(* Logix 5000 project; controller Hose_HP_Test_Rig_V1 vendor 1 type 14 code 149 rev 32.11; software revision 32.00; part 10 of 10 *)
(* tags used below, declared in another part *)
   INDV_LTEST_ON_STN4 : BOOL;
   ONS104 : BOOL;
   ONS4 : BOOL;
   TEST_INIT_DEL_STN4 : TIMER;
   AUTO_DOOR_OPEN_SEQ_STN4 : DINT;
   AUTO_TEST_ON_STN4 : BOOL;
   BOTTOM_CLAMP_SEQ_STN4 : DINT;
   BOTTOM_DECLAMP_SEQ_STN4 : DINT;
   CLR_ONS_STN4 : BOOL;
   CONS_CALB_ON_STN4 : BOOL;
   CONS_STS_STN1 : DINT;
   CONS_STS_STN2 : DINT;
   CONS_STS_STN3 : DINT;
   CONS_STS_STN4 : DINT;
   CONS_TEST_ON : BOOL;
   CYCLE_TIME_ACT_STN4 : REAL;
   DUMMIT : BOOL;
   FAIL_COUNT_RETEST : DINT;
   FAIL_COUNT_RETEST_STN2 : DINT;
   FAULTED_STN1 : BOOL;
   FAULTED_STN2 : BOOL;
   FAULTED_STN3 : BOOL;
   FAULTED_STN4 : BOOL;
   FP_ACCESS_OK : ALIAS FOR Local:2:I.Data.24;
   HP_SENSOR_SEL : BOOL;
   HP_STS_STN1 : DINT;
   HP_STS_STN2 : DINT;
   HP_STS_STN3 : DINT;
   HP_STS_STN4 : DINT;
   HP_TEST_ON : BOOL;
   INDV_CTEST_ON_STN4 : BOOL;
   INIT_STN4 : BOOL;
   MAIN_MENU : BOOL;
   MAIN_MENU_OFF : TIMER;
   OTHER_SENSOR_SEL : BOOL;
   PASS_COUNT_RETEST : DINT;
   PASS_COUNT_RETEST_STN2 : DINT;
   PASSED_STN4 : BOOL;
   PASSWORD_SET : DINT;
   RETEST : BOOL;
   RETEST_FAIL_COUNT : DINT;
   RETEST_ON_PROHIBIT : BOOL;
   RETEST_PASS_COUNT : DINT;
   RETEST_SET_COUNT : DINT;
   SCR_STS : DINT[6];
   SENS_CAL_SEL_BOTTOM_CLAMP : BOOL;
   SENS_CAL_SEL_MASTER : BOOL;
   SENS_CAL_SEL_STAMP : BOOL;
   SENS_CAL_SEL_TOP_CLAMP : BOOL;
   SENS_CALB_SEL_STN1 : BOOL;
   SENS_CALB_SEL_STN2 : BOOL;
   SENS_CALB_SEL_STN3 : BOOL;
   SENS_CALB_SEL_STN4 : BOOL;
   SEQ_NO_STN4 : DINT;
   STN1_TEST_STS : DINT;
   STN2_TEST_STS : DINT;
   STN3_TEST_STS : DINT;
   STN4_TEST_STS : DINT;
   STS : DINT;
   STS_OP_STN4 : DINT;
   TEST_ON_STN4 : BOOL;
   TOP_CLAMP_SEQ_STN4 : DINT;
   TS_STS_STN4 : DINT;
   USER_CHG : TIMER;
   VIEW_PARAM : BOOL;
   VIEW_PARAM_OFF : TIMER;
   WHICH_USER : INT;
(* MainProgram, continued *)

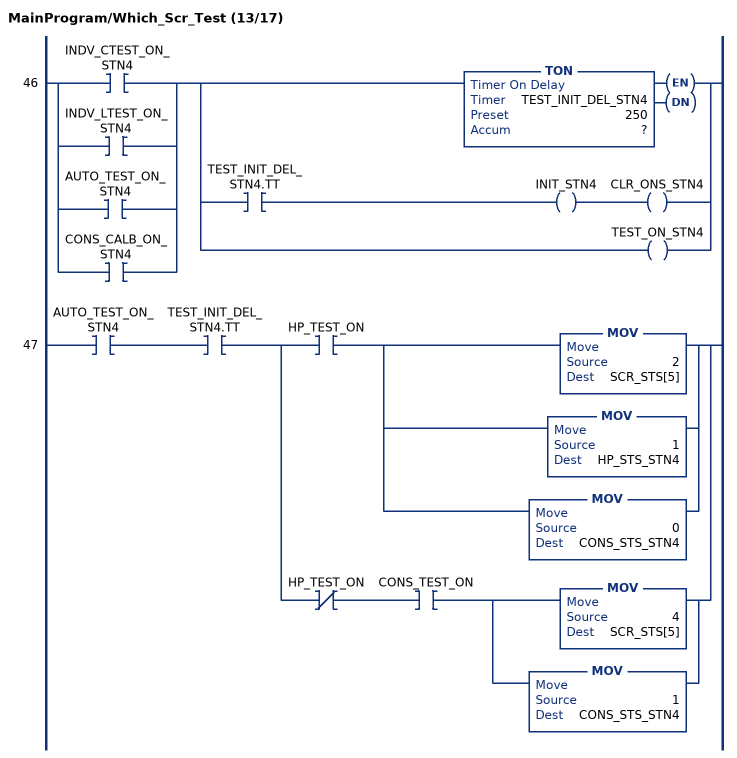
   [picture p174: MainProgram/Which_Scr_Test rungs 46-47]
   46: [XIC(INDV_CTEST_ON_STN4) ,XIC(INDV_LTEST_ON_STN4) ,XIC(AUTO_TEST_ON_STN4) ,XIC(CONS_CALB_ON_STN4) ][TON(TEST_INIT_DEL_STN4,?,?) ,XIC(TEST_INIT_DEL_STN4.TT) OTE(INIT_STN4) OTE(CLR_ONS_STN4) ,OTE(TEST_ON_STN4) ];
   47: XIC(AUTO_TEST_ON_STN4)XIC(TEST_INIT_DEL_STN4.TT)[XIC(HP_TEST_ON) [MOV(2,SCR_STS[5]) ,MOV(1,HP_STS_STN4) ,MOV(0,CONS_STS_STN4) ] ,XIO(HP_TEST_ON) XIC(CONS_TEST_ON) [MOV(4,SCR_STS[5]) ,MOV(1,CONS_STS_STN4) ] ];
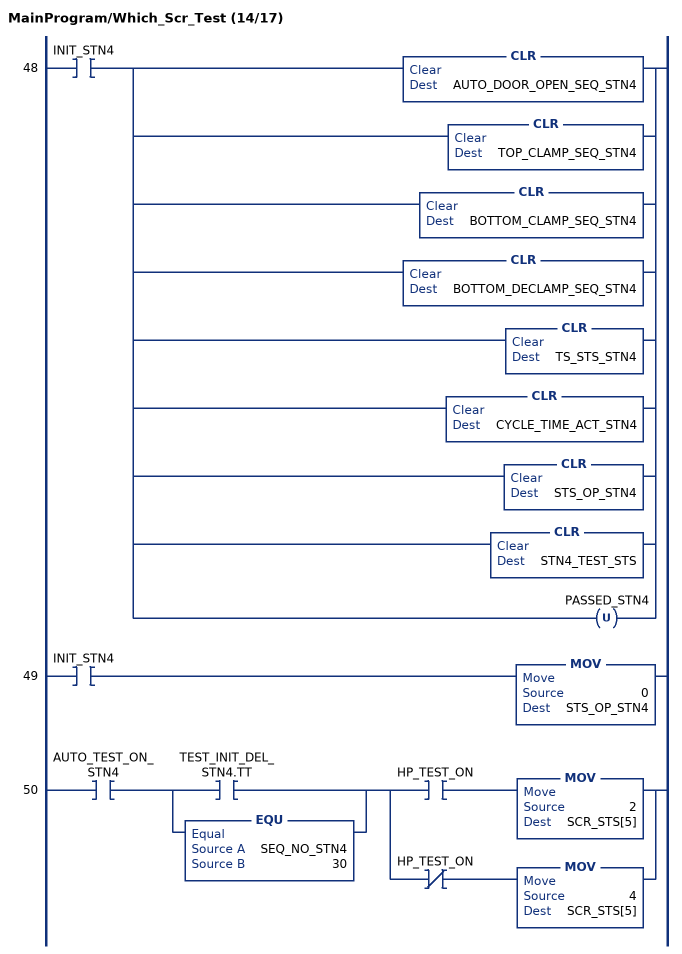
   48: XIC(INIT_STN4)[CLR(AUTO_DOOR_OPEN_SEQ_STN4) ,CLR(TOP_CLAMP_SEQ_STN4) ,CLR(BOTTOM_CLAMP_SEQ_STN4) ,CLR(BOTTOM_DECLAMP_SEQ_STN4) ,CLR(TS_STS_STN4) ,CLR(CYCLE_TIME_ACT_STN4) ,CLR(STS_OP_STN4) ,CLR(STN4_TEST_STS) ,OTU(PASSED_STN4) ];
   49: XIC(INIT_STN4)MOV(0,STS_OP_STN4);
   50: XIC(AUTO_TEST_ON_STN4)[XIC(TEST_INIT_DEL_STN4.TT) ,EQU(SEQ_NO_STN4,30) ][XIC(HP_TEST_ON) MOV(2,SCR_STS[5]) ,XIO(HP_TEST_ON) MOV(4,SCR_STS[5]) ];
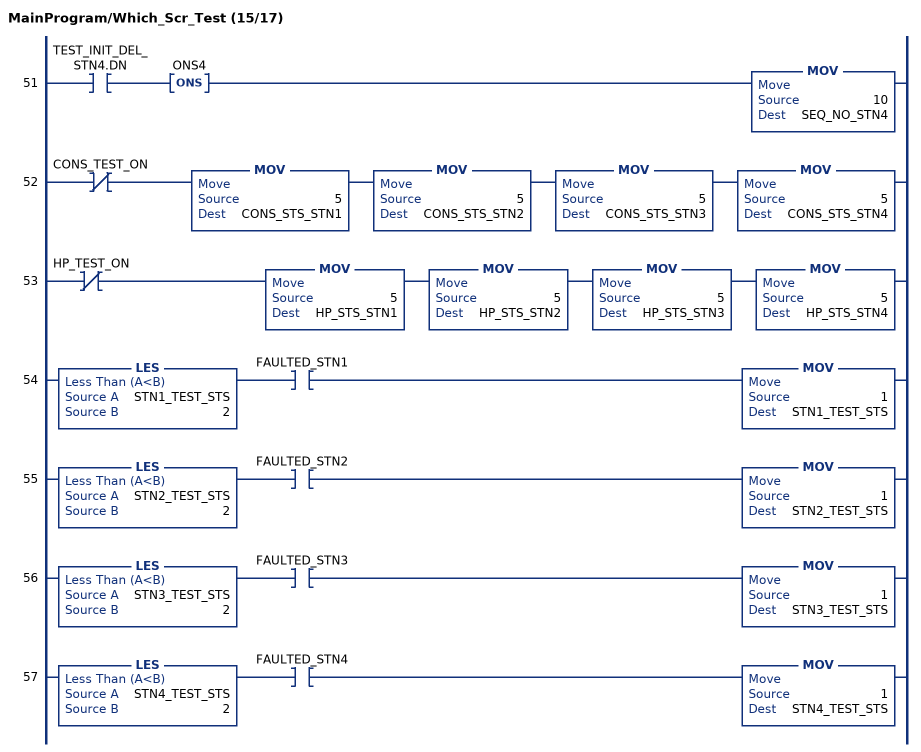
   51: XIC(TEST_INIT_DEL_STN4.DN)ONS(ONS4)MOV(10,SEQ_NO_STN4);
   52: XIO(CONS_TEST_ON)MOV(5,CONS_STS_STN1)MOV(5,CONS_STS_STN2)MOV(5,CONS_STS_STN3)MOV(5,CONS_STS_STN4);
   53: XIO(HP_TEST_ON)MOV(5,HP_STS_STN1)MOV(5,HP_STS_STN2)MOV(5,HP_STS_STN3)MOV(5,HP_STS_STN4);
   54: LES(STN1_TEST_STS,2)XIC(FAULTED_STN1)MOV(1,STN1_TEST_STS);
   55: LES(STN2_TEST_STS,2)XIC(FAULTED_STN2)MOV(1,STN2_TEST_STS);
   56: LES(STN3_TEST_STS,2)XIC(FAULTED_STN3)MOV(1,STN3_TEST_STS);
   57: LES(STN4_TEST_STS,2)XIC(FAULTED_STN4)MOV(1,STN4_TEST_STS);
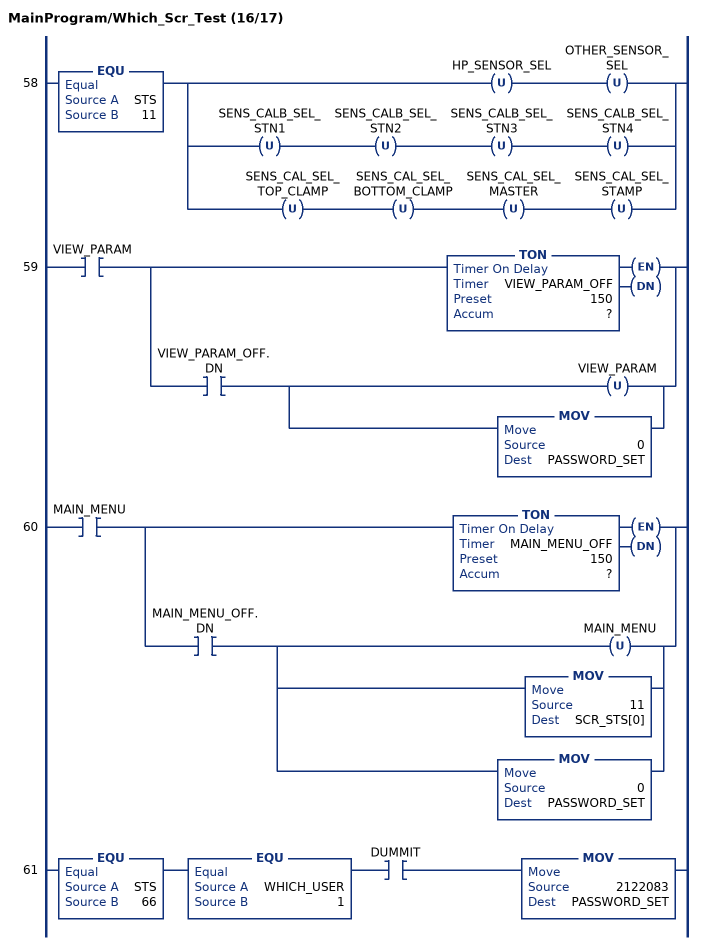
   58: EQU(STS,11)[OTU(HP_SENSOR_SEL) OTU(OTHER_SENSOR_SEL) ,OTU(SENS_CALB_SEL_STN1) OTU(SENS_CALB_SEL_STN2) OTU(SENS_CALB_SEL_STN3) OTU(SENS_CALB_SEL_STN4) ,OTU(SENS_CAL_SEL_TOP_CLAMP) OTU(SENS_CAL_SEL_BOTTOM_CLAMP) OTU(SENS_CAL_SEL_MASTER) OTU(SENS_CAL_SEL_STAMP) ];
   59: XIC(VIEW_PARAM)[TON(VIEW_PARAM_OFF,?,?) ,XIC(VIEW_PARAM_OFF.DN) [OTU(VIEW_PARAM) ,MOV(0,PASSWORD_SET) ] ];
   60: XIC(MAIN_MENU)[TON(MAIN_MENU_OFF,?,?) ,XIC(MAIN_MENU_OFF.DN) [OTU(MAIN_MENU) ,MOV(11,SCR_STS[0]) ,MOV(0,PASSWORD_SET) ] ];
   61: EQU(STS,66)EQU(WHICH_USER,1)XIC(DUMMIT)MOV(2122083,PASSWORD_SET);
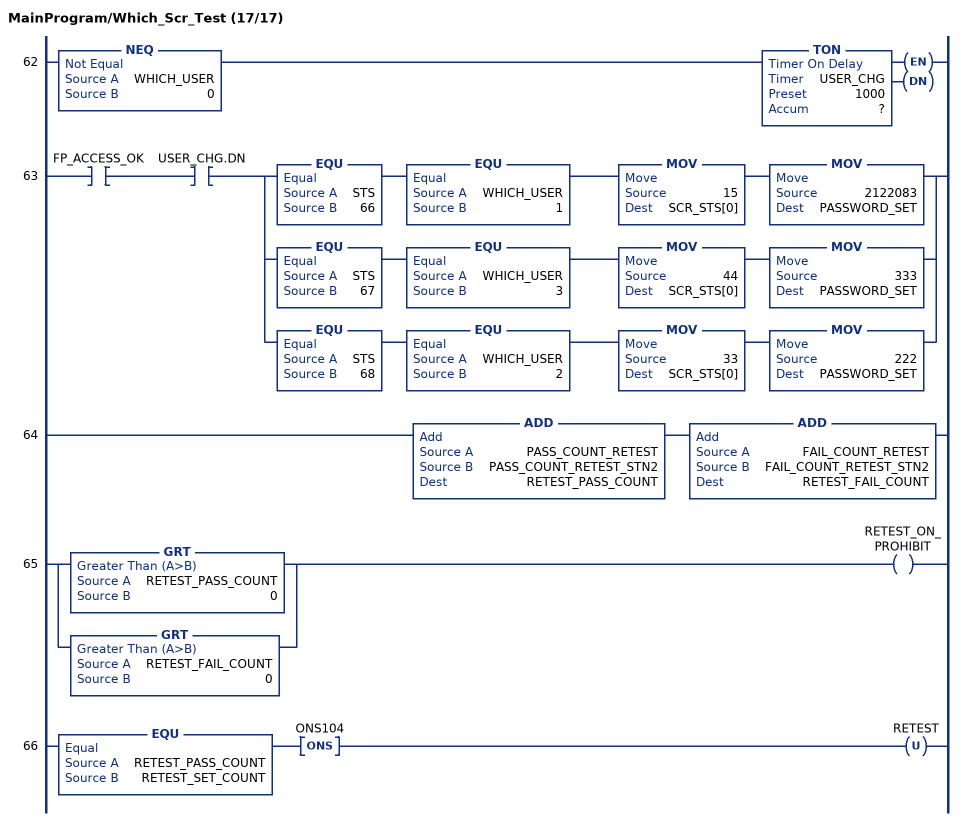
   62: NEQ(WHICH_USER,0)TON(USER_CHG,?,?);
   63: XIC(FP_ACCESS_OK)XIC(USER_CHG.DN)[EQU(STS,66) EQU(WHICH_USER,1) MOV(15,SCR_STS[0]) MOV(2122083,PASSWORD_SET) ,EQU(STS,67) EQU(WHICH_USER,3) MOV(44,SCR_STS[0]) MOV(333,PASSWORD_SET) ,EQU(STS,68) EQU(WHICH_USER,2) MOV(33,SCR_STS[0]) MOV(222,PASSWORD_SET) ];
   64: ADD(PASS_COUNT_RETEST,PASS_COUNT_RETEST_STN2,RETEST_PASS_COUNT)ADD(FAIL_COUNT_RETEST,FAIL_COUNT_RETEST_STN2,RETEST_FAIL_COUNT);
   65: [GRT(RETEST_PASS_COUNT,0) ,GRT(RETEST_FAIL_COUNT,0) ]OTE(RETEST_ON_PROHIBIT);
   66: EQU(RETEST_PASS_COUNT,RETEST_SET_COUNT)ONS(ONS104)OTU(RETEST);
END_ROUTINE
END_PROGRAM
